Yaskawa INFORM job: FMTV_HOOD_RIGHT.JBI

/JOB
//NAME FMTV_HOOD_RIGHT
//POS
///NPOS 63,0,0,0,0,0
///TOOL 0
///POSTYPE PULSE
///PULSE
C00000=-99132,-82437,-80579,-37363,-43577,-63256
C00001=-46769,-100860,-122047,-43256,-64895,-61432
C00002=7860,-119421,-92389,-49403,-100525,-59529
C00003=161067,-171476,-9214,-66644,112919,-54191
C00004=127681,-169179,32603,-76716,121253,-41393
C00005=127480,-167564,37485,-75908,120894,-40377
C00006=128238,-167981,36966,-75432,120772,-40429
C00007=128245,-168034,36807,-75458,120784,-40462
C00008=128505,-167812,37093,-75272,120728,-40452
C00009=128648,-167432,37533,-75164,120693,-40440
C00010=126697,-168878,36124,-76418,121149,-33116
C00011=126174,-169112,35108,-77822,119717,-32392
C00012=125377,-162918,42596,-81976,112780,-30182
C00013=124982,-157426,49873,-85897,107493,-27370
C00014=125327,-157980,52856,-87852,110302,-15431
C00015=125541,-159468,45925,-89349,111361,-17155
C00016=125542,-159467,45925,-89350,111361,-17154
C00017=126381,-155915,46234,-89949,111726,-25319
C00018=129648,-143875,56660,-88063,111237,-40735
C00019=130380,-142859,57867,-87524,111122,-40688
C00020=150971,-167078,30758,-67715,106901,-41414
C00021=150971,-167078,30758,-67715,106901,-41414
C00022=151684,-167308,30848,-67183,106743,-41350
C00023=152005,-166868,31450,-66944,106670,-41318
C00024=153108,-168657,32016,-65877,106029,-25214
C00025=153901,-169057,29614,-65600,106337,-25765
C00026=154760,-164431,39031,-65020,106279,-15545
C00027=153549,-161181,44960,-66528,110392,-7012
C00028=153549,-161181,44960,-66528,110392,-7012
C00029=154553,-161284,43353,-66124,110529,-7463
C00030=155048,-161072,41990,-66068,110777,-7911
C00031=155048,-161072,41990,-66068,110777,-7911
C00032=155048,-161072,41990,-66068,110777,-7911
C00033=155605,-160522,41049,-66128,111597,-8372
C00034=158297,-160955,38402,-64726,111685,-9070
C00035=158297,-160955,38402,-64726,111685,-9070
C00036=158297,-160955,38402,-64726,111685,-9070
C00037=159083,-162050,36450,-64345,111766,-9324
C00038=159975,-162134,35674,-63873,111806,-9540
C00039=158103,-162975,42240,-64270,107962,5225
C00040=159286,-160584,38772,-63655,114672,3761
C00041=158492,-163543,34726,-64393,115000,3514
C00042=158217,-165064,32754,-64666,115125,-52153
C00043=163556,-172483,-77551,-232337,81816,-52622
C00044=128292,-172357,-22942,-274601,81816,53651
C00045=110531,-157828,31930,-283347,100174,43304
C00046=110654,-140113,65199,-284464,98523,39166
C00047=110954,-137535,71523,-284520,98155,38158
C00048=121722,-134917,74068,-278158,100337,36097
C00049=121722,-134917,74068,-278158,100337,36097
C00050=123620,-135082,73251,-278187,100130,36255
C00051=124743,-135519,72545,-277634,100255,36102
C00052=125548,-136005,71843,-277230,100346,36005
C00053=126586,-136503,71202,-276513,100553,36032
C00054=128488,-138037,69336,-275187,100932,36095
C00055=133745,-143236,63128,-273519,103557,36466
C00056=142809,-151494,55153,-271023,108241,36528
C00057=149695,-157977,49778,-269274,111845,36281
C00058=153890,-161752,47432,-268506,114176,35886
C00059=162455,-169202,45107,-268131,119386,34294
C00060=163151,-172032,37869,-266439,119394,35673
C00061=163151,-172032,37869,-266439,119394,35673
C00062=164501,-173796,-97080,-262022,121018,-52705
//INST
///DATE 2023/03/28 15:40
///ATTR SC,RW
///GROUP1 RB1
NOP
MOVJ C00000 VJ=65.00  //FROM FRONT
MOVJ C00001 VJ=65.00
MOVJ C00002 VJ=65.00
MOVJ C00003 VJ=65.00
MOVL C00004 V=65.0  //UP TO
MOVL C00005 V=45.0  //INTO TOP
MOVL C00006 V=15.0
MOVC C00007 V=15.0
MOVC C00008 V=15.0
MOVC C00009 V=15.0
MOVL C00010 V=15.0
MOVL C00011 V=15.0
MOVL C00012 V=15.0
MOVL C00013 V=15.0
MOVL C00014 V=15.0
MOVL C00015 V=15.0
MOVC C00016 V=15.0
MOVC C00017 V=30.0
MOVC C00018 V=30.0
MOVL C00019 V=15.0
MOVL C00020 V=15.0
MOVC C00021 V=15.0
MOVC C00022 V=15.0
MOVC C00023 V=15.0
MOVL C00024 V=8.0
MOVL C00025 V=10.0
MOVL C00026 V=15.0
MOVL C00027 V=15.0
MOVC C00028 V=15.0
MOVC C00029 V=15.0
MOVC C00030 V=15.0
MOVL C00031 V=15.0
MOVC C00032 V=15.0
MOVC C00033 V=15.0
MOVC C00034 V=15.0
MOVL C00035 V=15.0
MOVC C00036 V=15.0
MOVC C00037 V=15.0
MOVC C00038 V=15.0
MOVL C00039 V=15.0
MOVL C00040 V=15.0
MOVL C00041 V=45.0  //OUT
MOVJ C00042 VJ=65.00
MOVJ C00043 VJ=65.00
MOVJ C00044 VJ=65.00
MOVL C00045 V=65.0  //ROTATE
MOVL C00046 V=65.0  //UP TO
MOVL C00047 V=15.0  //INTO BACK
MOVL C00048 V=15.0
MOVC C00049 V=15.0
MOVC C00050 V=15.0
MOVC C00051 V=15.0
MOVC C00052 V=15.0
MOVC C00053 V=15.0
MOVC C00054 V=15.0
MOVL C00055 V=15.0
MOVL C00056 V=15.0
MOVL C00057 V=15.0
MOVL C00058 V=15.0
MOVL C00059 V=15.0
MOVL C00060 V=45.0  //OUT
MOVJ C00061 VJ=65.00
MOVJ C00062 VJ=65.00  //CENTER
END
